PROGRAM CO_YPush_Error
VAR_IN_OUT
	Station		:structStationCtrl;
END_VAR

VAR
END_VAR

IF MC.ResetPressed THEN
	Station.SeqFaultWord := 0;
END_IF

(* 	Reserved Station.SeqFaultWord 
	= 1~49 for Major Fault
	= 100~149 for Origin Sequence Fault
	= 150~199 for Origin Width Adjust Sequence Fault
	= 200~299 for Auto Sequence Fault
	= 300~399 for misc fault listed on this page*)

Station.MajorFault := (Station.SeqFaultWord > 0) AND (Station.SeqFaultWord < 50);
Station.MinorFault := (Station.SeqFaultWord >= 100) OR Station.DeviceFault or E_PTC_BundleNOK;

END_PROGRAM

(* stored: Version 1.1.0.1, ProductVersion 3.1.4018.2
   POU CO_YPush_Error: Id {920255b3-b42f-48be-b292-97486ac60e8e}, SpecialFunc None *)
